FUNCTION_BLOCK CentralServer (* Composite Function Block Type that operates using Central Server *)
  (* Standard: 61499-2 *)
  (* Version 0.2, 2003-12-05, JHC, Rockwell Automation, Renamed from NEWCOMPFB. *)
  (* Version 0.1, 2002-01-08, JHC, Rockwell Automation, Added DLY FB as example. *)
  (* Version 0.0, 2000-05-27, JHC, Rockwell Automation *)
  (* Compiler header: package fb.rt.cs725; *)
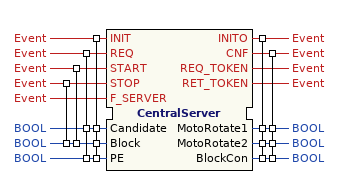
  EVENT_INPUT
    INIT WITH Candidate, Block, PE; (* Initialization Request *)
    REQ WITH Candidate, PE; (* Normal Execution Request *)
    START WITH Block;
    STOP WITH Block;
    F_SERVER;
  END_EVENT
  EVENT_OUTPUT
    INITO WITH MotoRotate1, MotoRotate2, BlockCon; (* Initialization Confirm *)
    CNF WITH MotoRotate1, MotoRotate2, BlockCon; (* Execution Confirmation *)
    REQ_TOKEN;
    RET_TOKEN;
  END_EVENT
  VAR_INPUT
    Candidate : BOOL;
    Block : BOOL;
    PE : BOOL;
  END_VAR
  VAR_OUTPUT
    MotoRotate1 : BOOL;
    MotoRotate2 : BOOL;
    BlockCon : BOOL;
  END_VAR
  FBS
    FC11 : ConveyorCTL(PE := 0, Block := 0, Candidate := 0);
    FC12 : CentralServerClient;
  END_FBS
  EVENT_CONNECTIONS
    INIT TO FC11.INIT;
    STOP TO FC12.CAS_STOP;
    START TO FC12.CAS_START;
    REQ TO FC12.REQ;
    FC12.CNF TO CNF;
    FC12.INITO TO INITO;
    FC11.INITO TO FC12.INIT;
    FC12.STOP TO FC11.CAS_STOP;
    FC12.START TO FC11.CAS_START;
    FC12.REQ_TOKEN TO REQ_TOKEN;
    FC12.RET_TOKEN TO RET_TOKEN;
    F_SERVER TO FC12.F_SERVER;
    REQ TO FC11.REQ;
  END_CONNECTIONS
  DATA_CONNECTIONS
    FC11.MotoRotate TO MotoRotate1;
    PE TO FC12.PE;
    Block TO FC12.Block;
    Candidate TO FC12.Candidate;
    FC12.MotoRotate TO MotoRotate2;
    FC12.BlockCon TO BlockCon;
  END_CONNECTIONS
END_FUNCTION_BLOCK
